TYPE E_DisconnectorPosition : 
(
    UNDEFINED := 0,
    OFF := 1,
    TURNING_ON := 2,
    ON := 3,
    TURNING_OFF := 4,
    FAULT := 5
);
END_TYPE

(* stored: Version 1.1.0.1, ProductVersion 3.1.4024.15
   EnumerationTextList E_DisconnectorPosition: Id {d87d6c25-eef3-46c6-9c9e-80da25ffd549} *)
